(* CoDeSys 2.3 export: displayFaultTest.py *)

(* POU Language, ST *)
PROGRAM Language
""")
outfile.write(declaration)
outfile.write( """END_VAR
""")
outfile.write("(*auto generated language definition file DO NOT alter manually *)\n")

for languageSet in languageSets:

    outfile.write( languageSets[languageSet])

outfile.close()
END_PROGRAM
